// TIA Portal V17 export
// export: Created 2025-03-05T08:00:04.7796525Z, ExportSetting WithDefaults, DisplayName Totally Integrated Automation Portal, DisplayVersion V17 Update 8, DisplayName TIA Portal Openness, DisplayVersion V17 Update 8, DisplayName TIA Portal Version Control Interface, DisplayVersion V17, DisplayName SINAMICS Startdrive Advanced, DisplayVersion V17 SP2, DisplayName SINAMICS Startdrive G110M, G120, G120C, G120D, G120P, G115D, DisplayVersion V17 SP2, DisplayName SINAMICS Startdrive G130, G150, S120, S150, SINAMICS MV, S210, DisplayVersion V17 SP2, DisplayName STEP 7 Professional, DisplayVersion V17 Update 8, DisplayName SINUMERIK ONE STEP 7 Toolbox, DisplayVersion V17 Update 12, DisplayName SINUMERIK 840D sl STEP 7 Toolbox, DisplayVersion V17 Update 12, DisplayName STEP 7 Safety, DisplayVersion V17 Update 6, DisplayName WinCC Advanced, DisplayVersion V17 Update 8
FUNCTION "FC2032_SINGLE_CYCLE" : Void   // FC2032, LAD
{ S7_Optimized_Access := 'FALSE' }
AUTHOR : ETXETAR
VERSION : 1.0
// stored: AutoNumber false, IsIECCheckEnabled false, SetENOAutomatically false, UDAEnableTagReadback false
   VAR CONSTANT
      FC_NUMBER : DInt := 2032;
   END_VAR
   VAR_TEMP   // added for the SCL form of the ladder/FBD networks
      _w1 : Bool;
      _w2 : Bool;
   END_VAR
BEGIN

REGION Network 1: CHANGE CYCLE GENERAL CONDITIONS
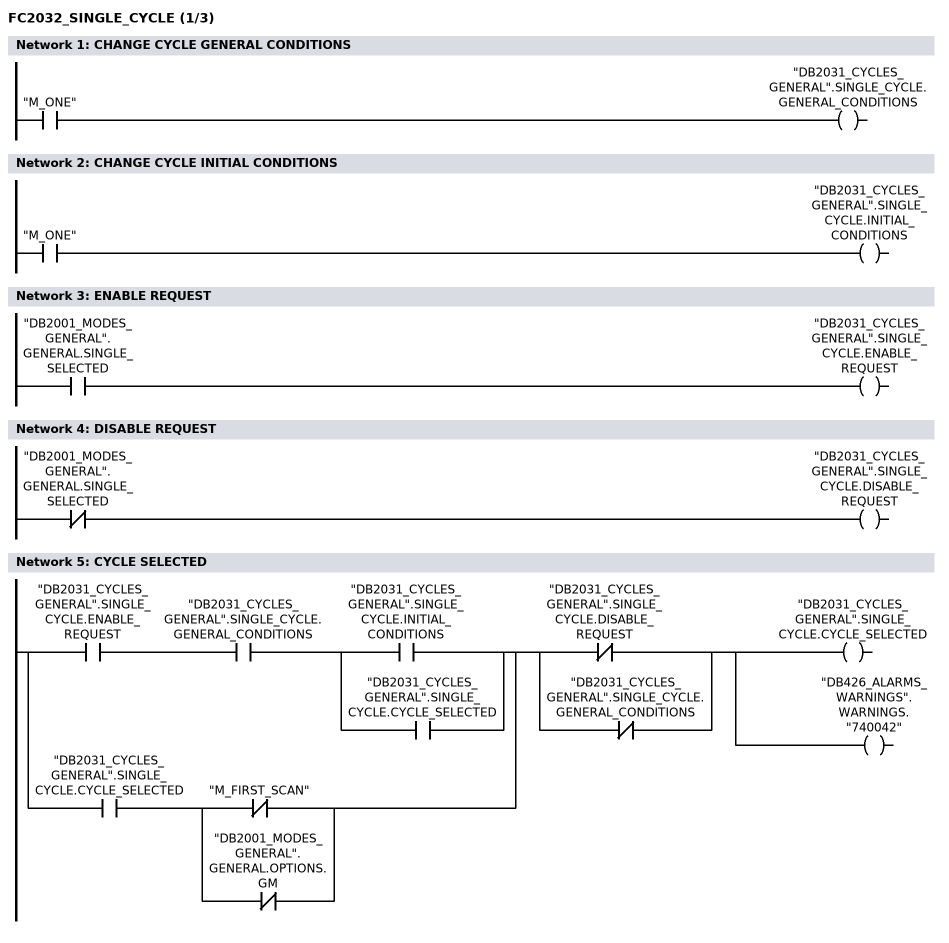
   RUNG wire#powerrail
      Contact( "M_ONE" )
      Coil( "DB2031_CYCLES_GENERAL".SINGLE_CYCLE.GENERAL_CONDITIONS )
   END_RUNG
   // the same network as SCL:
   "DB2031_CYCLES_GENERAL".SINGLE_CYCLE.GENERAL_CONDITIONS := "M_ONE";
END_REGION

REGION Network 2: CHANGE CYCLE INITIAL CONDITIONS
   RUNG wire#powerrail
      Contact( "M_ONE" )
      Coil( "DB2031_CYCLES_GENERAL".SINGLE_CYCLE.INITIAL_CONDITIONS )
   END_RUNG
   // the same network as SCL:
   "DB2031_CYCLES_GENERAL".SINGLE_CYCLE.INITIAL_CONDITIONS := "M_ONE";
END_REGION

REGION Network 3: ENABLE REQUEST
   RUNG wire#powerrail
      Contact( "DB2001_MODES_GENERAL".GENERAL.SINGLE_SELECTED )
      Coil( "DB2031_CYCLES_GENERAL".SINGLE_CYCLE.ENABLE_REQUEST )
   END_RUNG
   // the same network as SCL:
   "DB2031_CYCLES_GENERAL".SINGLE_CYCLE.ENABLE_REQUEST := "DB2001_MODES_GENERAL".GENERAL.SINGLE_SELECTED;
END_REGION

REGION Network 4: DISABLE REQUEST
   RUNG wire#powerrail
      I_Contact( "DB2001_MODES_GENERAL".GENERAL.SINGLE_SELECTED )
      Coil( "DB2031_CYCLES_GENERAL".SINGLE_CYCLE.DISABLE_REQUEST )
   END_RUNG
   // the same network as SCL:
   "DB2031_CYCLES_GENERAL".SINGLE_CYCLE.DISABLE_REQUEST := NOT "DB2001_MODES_GENERAL".GENERAL.SINGLE_SELECTED;
END_REGION

REGION Network 5: CYCLE SELECTED
   RUNG wire#powerrail
      Contact( "DB2031_CYCLES_GENERAL".SINGLE_CYCLE.ENABLE_REQUEST )
      Contact( "DB2031_CYCLES_GENERAL".SINGLE_CYCLE.GENERAL_CONDITIONS )
      wire#w1
      Contact( "DB2031_CYCLES_GENERAL".SINGLE_CYCLE.INITIAL_CONDITIONS )
      wire#w2
      I_Contact( "DB2031_CYCLES_GENERAL".SINGLE_CYCLE.DISABLE_REQUEST )
      wire#w4
      Coil( "DB2031_CYCLES_GENERAL".SINGLE_CYCLE.CYCLE_SELECTED )
   END_RUNG
   RUNG wire#w1
      Contact( "DB2031_CYCLES_GENERAL".SINGLE_CYCLE.CYCLE_SELECTED )
   END_RUNG wire#w2
   RUNG wire#powerrail
      Contact( "DB2031_CYCLES_GENERAL".SINGLE_CYCLE.CYCLE_SELECTED )
      wire#w3
      I_Contact( "M_FIRST_SCAN" )
   END_RUNG wire#w2
   RUNG wire#w3
      I_Contact( "DB2001_MODES_GENERAL".GENERAL.OPTIONS.GM )
   END_RUNG wire#w2
   RUNG wire#w2
      I_Contact( "DB2031_CYCLES_GENERAL".SINGLE_CYCLE.GENERAL_CONDITIONS )
   END_RUNG wire#w4
   RUNG wire#w4
      Coil( "DB426_ALARMS_WARNINGS".WARNINGS."740042" )
   END_RUNG
   // the same network as SCL:
   "DB2031_CYCLES_GENERAL".SINGLE_CYCLE.CYCLE_SELECTED := (("DB2031_CYCLES_GENERAL".SINGLE_CYCLE.ENABLE_REQUEST AND "DB2031_CYCLES_GENERAL".SINGLE_CYCLE.GENERAL_CONDITIONS AND ("DB2031_CYCLES_GENERAL".SINGLE_CYCLE.INITIAL_CONDITIONS OR "DB2031_CYCLES_GENERAL".SINGLE_CYCLE.CYCLE_SELECTED)) OR ("DB2031_CYCLES_GENERAL".SINGLE_CYCLE.CYCLE_SELECTED AND (NOT "M_FIRST_SCAN" OR NOT "DB2001_MODES_GENERAL".GENERAL.OPTIONS.GM))) AND (NOT "DB2031_CYCLES_GENERAL".SINGLE_CYCLE.DISABLE_REQUEST OR NOT "DB2031_CYCLES_GENERAL".SINGLE_CYCLE.GENERAL_CONDITIONS);
   "DB426_ALARMS_WARNINGS".WARNINGS."740042" := "DB2031_CYCLES_GENERAL".SINGLE_CYCLE.CYCLE_SELECTED;
END_REGION

REGION Network 6: CYCLE COMPLETED
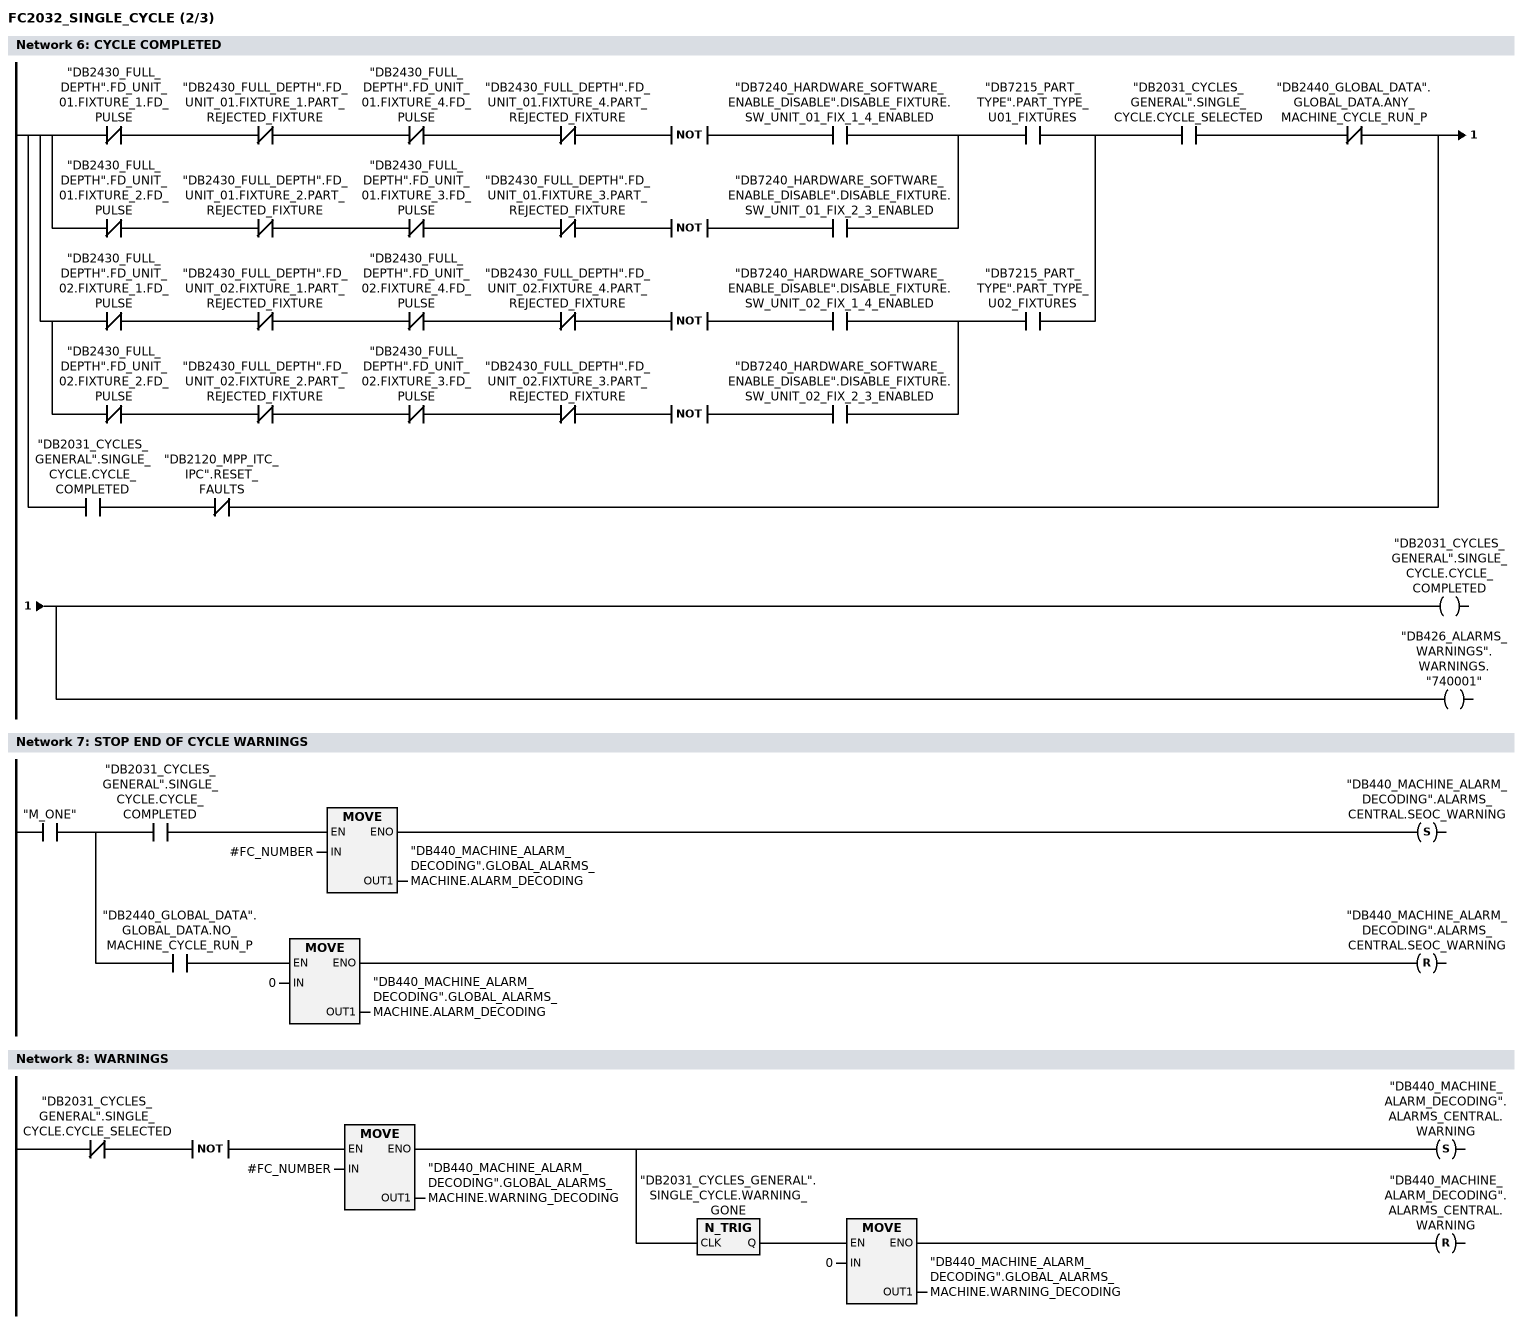
   RUNG wire#powerrail
      I_Contact( "DB2430_FULL_DEPTH".FD_UNIT_01.FIXTURE_1.FD_PULSE )
      I_Contact( "DB2430_FULL_DEPTH".FD_UNIT_01.FIXTURE_1.PART_REJECTED_FIXTURE )
      I_Contact( "DB2430_FULL_DEPTH".FD_UNIT_01.FIXTURE_4.FD_PULSE )
      I_Contact( "DB2430_FULL_DEPTH".FD_UNIT_01.FIXTURE_4.PART_REJECTED_FIXTURE )
      Not()
      Contact( "DB7240_HARDWARE_SOFTWARE_ENABLE_DISABLE".DISABLE_FIXTURE.SW_UNIT_01_FIX_1_4_ENABLED )
      wire#w1
      Contact( "DB7215_PART_TYPE".PART_TYPE_U01_FIXTURES )
      wire#w2
      Contact( "DB2031_CYCLES_GENERAL".SINGLE_CYCLE.CYCLE_SELECTED )
      I_Contact( "DB2440_GLOBAL_DATA".GLOBAL_DATA.ANY_MACHINE_CYCLE_RUN_P )
      wire#w4
      Coil( "DB2031_CYCLES_GENERAL".SINGLE_CYCLE.CYCLE_COMPLETED )
   END_RUNG
   RUNG wire#powerrail
      I_Contact( "DB2430_FULL_DEPTH".FD_UNIT_01.FIXTURE_2.FD_PULSE )
      I_Contact( "DB2430_FULL_DEPTH".FD_UNIT_01.FIXTURE_2.PART_REJECTED_FIXTURE )
      I_Contact( "DB2430_FULL_DEPTH".FD_UNIT_01.FIXTURE_3.FD_PULSE )
      I_Contact( "DB2430_FULL_DEPTH".FD_UNIT_01.FIXTURE_3.PART_REJECTED_FIXTURE )
      Not()
      Contact( "DB7240_HARDWARE_SOFTWARE_ENABLE_DISABLE".DISABLE_FIXTURE.SW_UNIT_01_FIX_2_3_ENABLED )
   END_RUNG wire#w1
   RUNG wire#powerrail
      I_Contact( "DB2430_FULL_DEPTH".FD_UNIT_02.FIXTURE_1.FD_PULSE )
      I_Contact( "DB2430_FULL_DEPTH".FD_UNIT_02.FIXTURE_1.PART_REJECTED_FIXTURE )
      I_Contact( "DB2430_FULL_DEPTH".FD_UNIT_02.FIXTURE_4.FD_PULSE )
      I_Contact( "DB2430_FULL_DEPTH".FD_UNIT_02.FIXTURE_4.PART_REJECTED_FIXTURE )
      Not()
      Contact( "DB7240_HARDWARE_SOFTWARE_ENABLE_DISABLE".DISABLE_FIXTURE.SW_UNIT_02_FIX_1_4_ENABLED )
      wire#w3
      Contact( "DB7215_PART_TYPE".PART_TYPE_U02_FIXTURES )
   END_RUNG wire#w2
   RUNG wire#powerrail
      I_Contact( "DB2430_FULL_DEPTH".FD_UNIT_02.FIXTURE_2.FD_PULSE )
      I_Contact( "DB2430_FULL_DEPTH".FD_UNIT_02.FIXTURE_2.PART_REJECTED_FIXTURE )
      I_Contact( "DB2430_FULL_DEPTH".FD_UNIT_02.FIXTURE_3.FD_PULSE )
      I_Contact( "DB2430_FULL_DEPTH".FD_UNIT_02.FIXTURE_3.PART_REJECTED_FIXTURE )
      Not()
      Contact( "DB7240_HARDWARE_SOFTWARE_ENABLE_DISABLE".DISABLE_FIXTURE.SW_UNIT_02_FIX_2_3_ENABLED )
   END_RUNG wire#w3
   RUNG wire#powerrail
      Contact( "DB2031_CYCLES_GENERAL".SINGLE_CYCLE.CYCLE_COMPLETED )
      I_Contact( "DB2120_MPP_ITC_IPC".RESET_FAULTS )
   END_RUNG wire#w4
   RUNG wire#w4
      Coil( "DB426_ALARMS_WARNINGS".WARNINGS."740001" )
   END_RUNG
   // the same network as SCL:
   "DB2031_CYCLES_GENERAL".SINGLE_CYCLE.CYCLE_COMPLETED := (((((NOT (NOT "DB2430_FULL_DEPTH".FD_UNIT_01.FIXTURE_1.FD_PULSE AND NOT "DB2430_FULL_DEPTH".FD_UNIT_01.FIXTURE_1.PART_REJECTED_FIXTURE AND NOT "DB2430_FULL_DEPTH".FD_UNIT_01.FIXTURE_4.FD_PULSE AND NOT "DB2430_FULL_DEPTH".FD_UNIT_01.FIXTURE_4.PART_REJECTED_FIXTURE) AND "DB7240_HARDWARE_SOFTWARE_ENABLE_DISABLE".DISABLE_FIXTURE.SW_UNIT_01_FIX_1_4_ENABLED) OR (NOT (NOT "DB2430_FULL_DEPTH".FD_UNIT_01.FIXTURE_2.FD_PULSE AND NOT "DB2430_FULL_DEPTH".FD_UNIT_01.FIXTURE_2.PART_REJECTED_FIXTURE AND NOT "DB2430_FULL_DEPTH".FD_UNIT_01.FIXTURE_3.FD_PULSE AND NOT "DB2430_FULL_DEPTH".FD_UNIT_01.FIXTURE_3.PART_REJECTED_FIXTURE) AND "DB7240_HARDWARE_SOFTWARE_ENABLE_DISABLE".DISABLE_FIXTURE.SW_UNIT_01_FIX_2_3_ENABLED)) AND "DB7215_PART_TYPE".PART_TYPE_U01_FIXTURES) OR (((NOT (NOT "DB2430_FULL_DEPTH".FD_UNIT_02.FIXTURE_1.FD_PULSE AND NOT "DB2430_FULL_DEPTH".FD_UNIT_02.FIXTURE_1.PART_REJECTED_FIXTURE AND NOT "DB2430_FULL_DEPTH".FD_UNIT_02.FIXTURE_4.FD_PULSE AND NOT "DB2430_FULL_DEPTH".FD_UNIT_02.FIXTURE_4.PART_REJECTED_FIXTURE) AND "DB7240_HARDWARE_SOFTWARE_ENABLE_DISABLE".DISABLE_FIXTURE.SW_UNIT_02_FIX_1_4_ENABLED) OR (NOT (NOT "DB2430_FULL_DEPTH".FD_UNIT_02.FIXTURE_2.FD_PULSE AND NOT "DB2430_FULL_DEPTH".FD_UNIT_02.FIXTURE_2.PART_REJECTED_FIXTURE AND NOT "DB2430_FULL_DEPTH".FD_UNIT_02.FIXTURE_3.FD_PULSE AND NOT "DB2430_FULL_DEPTH".FD_UNIT_02.FIXTURE_3.PART_REJECTED_FIXTURE) AND "DB7240_HARDWARE_SOFTWARE_ENABLE_DISABLE".DISABLE_FIXTURE.SW_UNIT_02_FIX_2_3_ENABLED)) AND "DB7215_PART_TYPE".PART_TYPE_U02_FIXTURES)) AND "DB2031_CYCLES_GENERAL".SINGLE_CYCLE.CYCLE_SELECTED AND NOT "DB2440_GLOBAL_DATA".GLOBAL_DATA.ANY_MACHINE_CYCLE_RUN_P) OR ("DB2031_CYCLES_GENERAL".SINGLE_CYCLE.CYCLE_COMPLETED AND NOT "DB2120_MPP_ITC_IPC".RESET_FAULTS);
   "DB426_ALARMS_WARNINGS".WARNINGS."740001" := "DB2031_CYCLES_GENERAL".SINGLE_CYCLE.CYCLE_COMPLETED;
END_REGION

REGION Network 7: STOP END OF CYCLE WARNINGS
   RUNG wire#powerrail
      Contact( "M_ONE" )
      wire#w1
      Contact( "DB2031_CYCLES_GENERAL".SINGLE_CYCLE.CYCLE_COMPLETED )
      { S7_GenerateENO := "TRUE" } Move(in := #FC_NUMBER, out1 => "DB440_MACHINE_ALARM_DECODING".GLOBAL_ALARMS_MACHINE.ALARM_DECODING)
      S_Coil( "DB440_MACHINE_ALARM_DECODING".ALARMS_CENTRAL.SEOC_WARNING )
   END_RUNG
   RUNG wire#w1
      Contact( "DB2440_GLOBAL_DATA".GLOBAL_DATA.NO_MACHINE_CYCLE_RUN_P )
      { S7_GenerateENO := "TRUE" } Move(in := 0, out1 => "DB440_MACHINE_ALARM_DECODING".GLOBAL_ALARMS_MACHINE.ALARM_DECODING)
      R_Coil( "DB440_MACHINE_ALARM_DECODING".ALARMS_CENTRAL.SEOC_WARNING )
   END_RUNG
   // the same network as SCL:
   // ENO of a box is taken as its EN; it also drops when the box reports an error
   IF "M_ONE" AND "DB2031_CYCLES_GENERAL".SINGLE_CYCLE.CYCLE_COMPLETED THEN
       "DB440_MACHINE_ALARM_DECODING".GLOBAL_ALARMS_MACHINE.ALARM_DECODING := #FC_NUMBER;
       "DB440_MACHINE_ALARM_DECODING".ALARMS_CENTRAL.SEOC_WARNING := TRUE;
   END_IF;
   IF "M_ONE" AND "DB2440_GLOBAL_DATA".GLOBAL_DATA.NO_MACHINE_CYCLE_RUN_P THEN
       "DB440_MACHINE_ALARM_DECODING".GLOBAL_ALARMS_MACHINE.ALARM_DECODING := 0;
       "DB440_MACHINE_ALARM_DECODING".ALARMS_CENTRAL.SEOC_WARNING := FALSE;
   END_IF;
END_REGION

REGION Network 8: WARNINGS
   RUNG wire#powerrail
      I_Contact( "DB2031_CYCLES_GENERAL".SINGLE_CYCLE.CYCLE_SELECTED )
      Not()
      Move(in := #FC_NUMBER, out1 => "DB440_MACHINE_ALARM_DECODING".GLOBAL_ALARMS_MACHINE.WARNING_DECODING)
      wire#w1
      S_Coil( "DB440_MACHINE_ALARM_DECODING".ALARMS_CENTRAL.WARNING )
   END_RUNG
   RUNG wire#w1
      N_Trig( "DB2031_CYCLES_GENERAL".SINGLE_CYCLE.WARNING_GONE )
      Move(in := 0, out1 => "DB440_MACHINE_ALARM_DECODING".GLOBAL_ALARMS_MACHINE.WARNING_DECODING)
      R_Coil( "DB440_MACHINE_ALARM_DECODING".ALARMS_CENTRAL.WARNING )
   END_RUNG
   // the same network as SCL:
   #_w1 := NOT (NOT "DB2031_CYCLES_GENERAL".SINGLE_CYCLE.CYCLE_SELECTED);
   IF #_w1 THEN
       "DB440_MACHINE_ALARM_DECODING".GLOBAL_ALARMS_MACHINE.WARNING_DECODING := #FC_NUMBER;
       "DB440_MACHINE_ALARM_DECODING".ALARMS_CENTRAL.WARNING := TRUE;
   END_IF;
   #_w2 := NOT #_w1 AND "DB2031_CYCLES_GENERAL".SINGLE_CYCLE.WARNING_GONE;   // falling edge
   "DB2031_CYCLES_GENERAL".SINGLE_CYCLE.WARNING_GONE := #_w1;
   IF #_w2 THEN
       "DB440_MACHINE_ALARM_DECODING".GLOBAL_ALARMS_MACHINE.WARNING_DECODING := 0;
       "DB440_MACHINE_ALARM_DECODING".ALARMS_CENTRAL.WARNING := FALSE;
   END_IF;
END_REGION

REGION Network 9: CHANGE CYCLE GENERAL CONDITIONS HELP
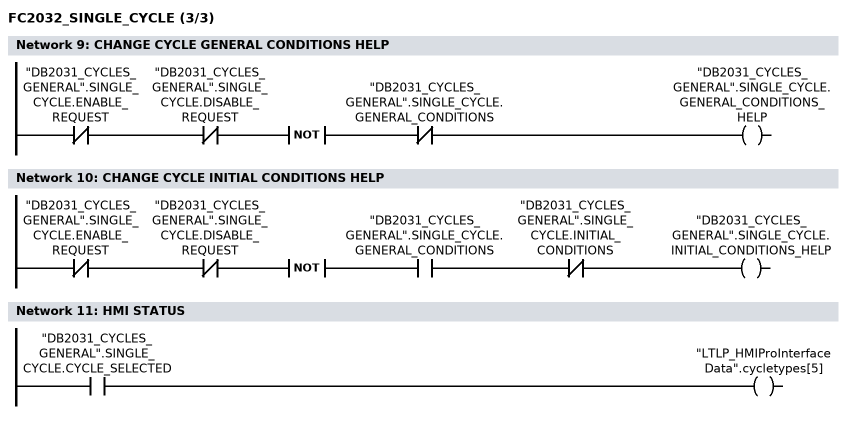
   RUNG wire#powerrail
      I_Contact( "DB2031_CYCLES_GENERAL".SINGLE_CYCLE.ENABLE_REQUEST )
      I_Contact( "DB2031_CYCLES_GENERAL".SINGLE_CYCLE.DISABLE_REQUEST )
      Not()
      I_Contact( "DB2031_CYCLES_GENERAL".SINGLE_CYCLE.GENERAL_CONDITIONS )
      Coil( "DB2031_CYCLES_GENERAL".SINGLE_CYCLE.GENERAL_CONDITIONS_HELP )
   END_RUNG
   // the same network as SCL:
   "DB2031_CYCLES_GENERAL".SINGLE_CYCLE.GENERAL_CONDITIONS_HELP := NOT (NOT "DB2031_CYCLES_GENERAL".SINGLE_CYCLE.ENABLE_REQUEST AND NOT "DB2031_CYCLES_GENERAL".SINGLE_CYCLE.DISABLE_REQUEST) AND NOT "DB2031_CYCLES_GENERAL".SINGLE_CYCLE.GENERAL_CONDITIONS;
END_REGION

REGION Network 10: CHANGE CYCLE INITIAL CONDITIONS HELP
   RUNG wire#powerrail
      I_Contact( "DB2031_CYCLES_GENERAL".SINGLE_CYCLE.ENABLE_REQUEST )
      I_Contact( "DB2031_CYCLES_GENERAL".SINGLE_CYCLE.DISABLE_REQUEST )
      Not()
      Contact( "DB2031_CYCLES_GENERAL".SINGLE_CYCLE.GENERAL_CONDITIONS )
      I_Contact( "DB2031_CYCLES_GENERAL".SINGLE_CYCLE.INITIAL_CONDITIONS )
      Coil( "DB2031_CYCLES_GENERAL".SINGLE_CYCLE.INITIAL_CONDITIONS_HELP )
   END_RUNG
   // the same network as SCL:
   "DB2031_CYCLES_GENERAL".SINGLE_CYCLE.INITIAL_CONDITIONS_HELP := NOT (NOT "DB2031_CYCLES_GENERAL".SINGLE_CYCLE.ENABLE_REQUEST AND NOT "DB2031_CYCLES_GENERAL".SINGLE_CYCLE.DISABLE_REQUEST) AND "DB2031_CYCLES_GENERAL".SINGLE_CYCLE.GENERAL_CONDITIONS AND NOT "DB2031_CYCLES_GENERAL".SINGLE_CYCLE.INITIAL_CONDITIONS;
END_REGION

REGION Network 11: HMI STATUS
   RUNG wire#powerrail
      Contact( "DB2031_CYCLES_GENERAL".SINGLE_CYCLE.CYCLE_SELECTED )
      Coil( "LTLP_HMIProInterfaceData".cycletypes[5] )
   END_RUNG
   // the same network as SCL:
   "LTLP_HMIProInterfaceData".cycletypes[5] := "DB2031_CYCLES_GENERAL".SINGLE_CYCLE.CYCLE_SELECTED;
END_REGION
END_FUNCTION
